TYPE ST_ModbusRegister :
STRUCT
	Reg_Adress: UDINT;
	Num_Bytes: INT;
	Value_Type: E_ModbusDataType;
	Description: STRING;
	AccessType: E_AccessType;
	Value: ARRAY[1..4] OF WORD;
END_STRUCT
END_TYPE

(* stored: Version 1.1.0.1, ProductVersion 3.1.4024.12
   DUT ST_ModbusRegister: Id {89f224b5-0136-4cd5-8fe4-b1eb3c939a54} *)
